(* delete old files and delete oldest files if number of files exceeds specified number *)
PROGRAM C09_MaintainFolders
VAR
	tArchiveCheck				: TIME := t#4s;
	fbMaintainArchive			: FB_PulseGenerator;
	tDeleteTimeCheck			: TIME := t#20m;
	fbMaintainDeleteTime		: FB_PulseGenerator;
	tClearProcessFolders		: TIME := T#500MS;
	tofClearProcessFolders		: TOF;
	
	nActivateBitWord			: DWORD; (* if index increase 32 bits it is necceasry to declar 64 bits var like LREAL;*)

	aMaintainFolders			: ARRAY[1..18] OF NT_StartProcess;
	aManualMaintain				: ARRAY[1..18] OF BOOL;

	fbMoveCHMToArchive			: FB_CHM_MoveToArchive;
	bZipCHMArchive				: BOOL;
	rtrigZipAfetrPassthrough	: R_TRIG;
	bManualZip					: BOOL;
	
(********************************************************************************
cMETS_CORE_FOLDERS					: ARRAY[1..cSYSTEM_FOLDER_LIMIT] OF T_FolderName :=[
			(*01*)'CHM\',		(*02*)'CHM\Archive\',		(*03*)'CHM\Error\',		(*04*)'CHM\OK\',		(*05*)'CHM\Commissioning_Mode\',	(*06*)'CHM\Restore\',
			(*07*)'PCM\',		(*08*)'PCM\Archive\',		(*09*)'PCM\Error\',		(*10*)'PCM\Incoming\',
			(*11*)'Settings\',	(*12*)'Settings\Backups\',	(*13*)'Settings\Recipe\',
			(*14*)'Cameras\',
			(*15*)'Printers\',	(*16*)'Printers\Templates'];
			
cMETS_AUX_FOLDERS					: ARRAY[1..cSYSTEM_FOLDER_LIMIT] OF T_FolderName :=[
			(*01*)'CAC\',		(*02*)'CAC\Archive\',		(*03*)'CAC\Error\',		(*04*)'CAC\Restored\',
			(*05*)'OAC\',		(*06*)'OAC\Error\',			(*07*)'OAC\Empty\',
			(*08*)'OCV\',		(*09*)'OCV\Error\',			(*10*)'OCV\Empty\',
			(*11*)'SystemLog\',
			(*12*)'ArchiveDB\',
			(*13*)'BridgeApp\Bridge_Core\',
			(*14*)'LoggerApp\Service\',
			(*15*)'WebHMI\',
			(*16*)'DeleteArchiveTool\'];

*************************************************************************************)
(********************************************************************************
Delete Items
	DeleteItem <path> <filesToKeep> [createLog] [deleteDirs] [dirsToKeep]
	path: Directory path
	filesToKeep: Number OF files TO RETAIN
	createLog: (Optional) Boolean to enable logging
	deleteDirs: (Optional) Boolean to include directories
	dirsToKeep: (Optional) Number of directories to retain

Delete by Time
	DeleteTime <path> <fileAge> [createLog] [deleteDirs] [ageUnit]
	path: Directory path
	fileAge: Maximum age of files to retain
	createLog: (Optional) Boolean to enable logging
	deleteDirs: (Optional) Boolean to include inside directories for file search
	ageUnit: (Optional) Time unit for age values (Day/Hour/Minute), defaults to Day

Archive
	Archive <chmArchiveFolder> <lastArchiveDateName> [createLog]
	chmArchiveFolder: Archive folder path
	lastArchiveDateName: Last archive date identifier
	createLog: (Optional) Boolean TO enable logging
*************************************************************************************)
END_VAR

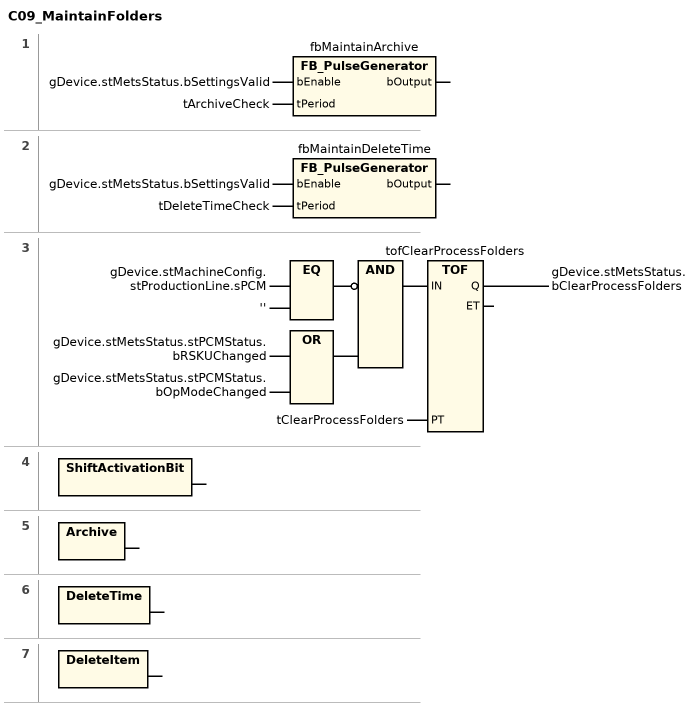
// NETWORK 1
fbMaintainArchive(bEnable := gDevice.stMetsStatus.bSettingsValid, tPeriod := tArchiveCheck); // FB_PulseGenerator

// NETWORK 2
fbMaintainDeleteTime(bEnable := gDevice.stMetsStatus.bSettingsValid, tPeriod := tDeleteTimeCheck); // FB_PulseGenerator

// NETWORK 3
tofClearProcessFolders(IN := NOT (gDevice.stMachineConfig.stProductionLine.sPCM = '') AND (gDevice.stMetsStatus.stPCMStatus.bRSKUChanged OR gDevice.stMetsStatus.stPCMStatus.bOpModeChanged), PT := tClearProcessFolders); // TOF
gDevice.stMetsStatus.bClearProcessFolders := tofClearProcessFolders.Q;

// NETWORK 4
ShiftActivationBit();

// NETWORK 5
Archive();

// NETWORK 6
DeleteTime();

// NETWORK 7
DeleteItem();

ACTION Archive:
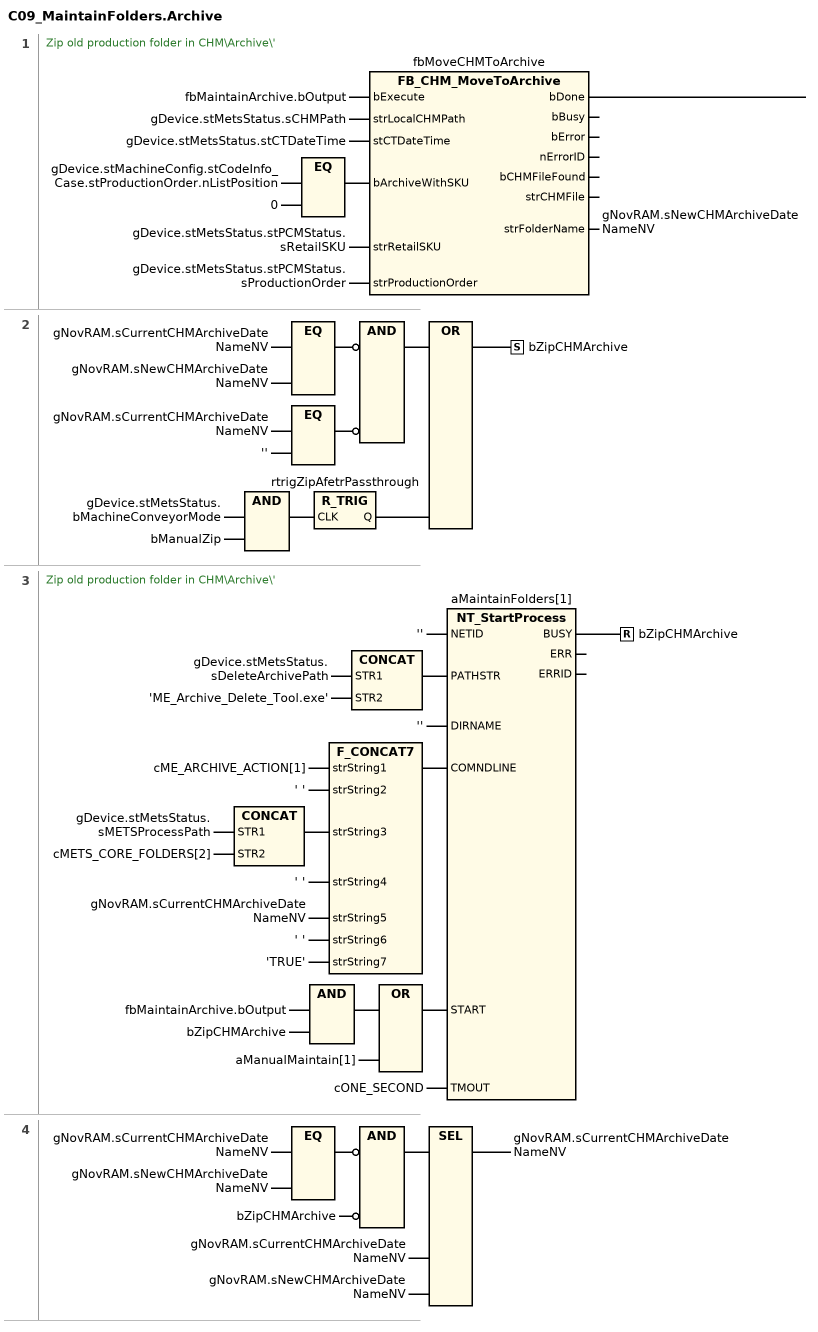
// NETWORK 1
// 					Zip old production folder in CHM\Archive\'
//
//
fbMoveCHMToArchive(
    bExecute := fbMaintainArchive.bOutput,
    strLocalCHMPath := gDevice.stMetsStatus.sCHMPath,
    stCTDateTime := gDevice.stMetsStatus.stCTDateTime,
    bArchiveWithSKU := gDevice.stMachineConfig.stCodeInfo_Case.stProductionOrder.nListPosition = 0,
    strRetailSKU := gDevice.stMetsStatus.stPCMStatus.sRetailSKU,
    strProductionOrder := gDevice.stMetsStatus.stPCMStatus.sProductionOrder,
    strFolderName => gNovRAM.sNewCHMArchiveDateNameNV); // FB_CHM_MoveToArchive

// NETWORK 2
rtrigZipAfetrPassthrough(CLK := gDevice.stMetsStatus.bMachineConveyorMode AND bManualZip); // R_TRIG
bZipCHMArchive S= NOT (gNovRAM.sCurrentCHMArchiveDateNameNV = gNovRAM.sNewCHMArchiveDateNameNV) AND NOT (gNovRAM.sCurrentCHMArchiveDateNameNV = '') OR rtrigZipAfetrPassthrough.Q;

// NETWORK 3
// Zip old production folder in CHM\Archive\'
aMaintainFolders[1](
    NETID := '',
    PATHSTR := CONCAT(STR1 := gDevice.stMetsStatus.sDeleteArchivePath, STR2 := 'ME_Archive_Delete_Tool.exe'),
    DIRNAME := '',
    COMNDLINE := F_CONCAT7(strString1 := cME_ARCHIVE_ACTION[1], strString2 := ' ', strString3 := CONCAT(STR1 := gDevice.stMetsStatus.sMETSProcessPath, STR2 := cMETS_CORE_FOLDERS[2]), strString4 := ' ', strString5 := gNovRAM.sCurrentCHMArchiveDateNameNV, strString6 := ' ', strString7 := 'TRUE'),
    START := fbMaintainArchive.bOutput AND bZipCHMArchive OR aManualMaintain[1],
    TMOUT := cONE_SECOND); // NT_StartProcess
bZipCHMArchive R= aMaintainFolders[1].BUSY;

// NETWORK 4
gNovRAM.sCurrentCHMArchiveDateNameNV := SEL(NOT (gNovRAM.sCurrentCHMArchiveDateNameNV = gNovRAM.sNewCHMArchiveDateNameNV) AND NOT bZipCHMArchive, gNovRAM.sCurrentCHMArchiveDateNameNV, gNovRAM.sNewCHMArchiveDateNameNV);
END_ACTION

ACTION DeleteItem:
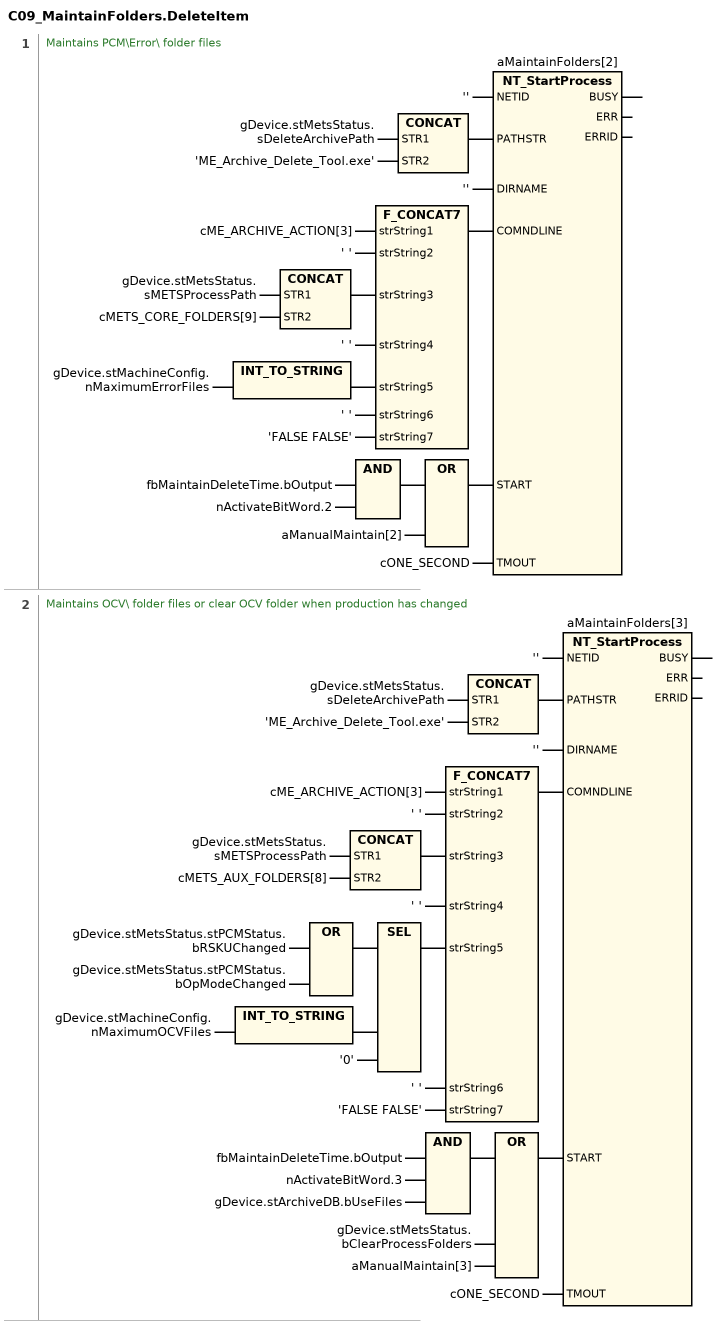
// NETWORK 1
// Maintains PCM\Error\ folder files
aMaintainFolders[2](
    NETID := '',
    PATHSTR := CONCAT(STR1 := gDevice.stMetsStatus.sDeleteArchivePath, STR2 := 'ME_Archive_Delete_Tool.exe'),
    DIRNAME := '',
    COMNDLINE := F_CONCAT7(strString1 := cME_ARCHIVE_ACTION[3], strString2 := ' ', strString3 := CONCAT(STR1 := gDevice.stMetsStatus.sMETSProcessPath, STR2 := cMETS_CORE_FOLDERS[9]), strString4 := ' ', strString5 := INT_TO_STRING(gDevice.stMachineConfig.nMaximumErrorFiles), strString6 := ' ', strString7 := 'FALSE FALSE'),
    START := fbMaintainDeleteTime.bOutput AND nActivateBitWord.2 OR aManualMaintain[2],
    TMOUT := cONE_SECOND); // NT_StartProcess

// NETWORK 2
// Maintains OCV\ folder files or clear OCV folder when production has changed
aMaintainFolders[3](
    NETID := '',
    PATHSTR := CONCAT(STR1 := gDevice.stMetsStatus.sDeleteArchivePath, STR2 := 'ME_Archive_Delete_Tool.exe'),
    DIRNAME := '',
    COMNDLINE := F_CONCAT7(strString1 := cME_ARCHIVE_ACTION[3], strString2 := ' ', strString3 := CONCAT(STR1 := gDevice.stMetsStatus.sMETSProcessPath, STR2 := cMETS_AUX_FOLDERS[8]), strString4 := ' ', strString5 := SEL(gDevice.stMetsStatus.stPCMStatus.bRSKUChanged OR gDevice.stMetsStatus.stPCMStatus.bOpModeChanged, INT_TO_STRING(gDevice.stMachineConfig.nMaximumOCVFiles), '0'), strString6 := ' ', strString7 := 'FALSE FALSE'),
    START := fbMaintainDeleteTime.bOutput AND nActivateBitWord.3 AND gDevice.stArchiveDB.bUseFiles OR gDevice.stMetsStatus.bClearProcessFolders OR aManualMaintain[3],
    TMOUT := cONE_SECOND); // NT_StartProcess

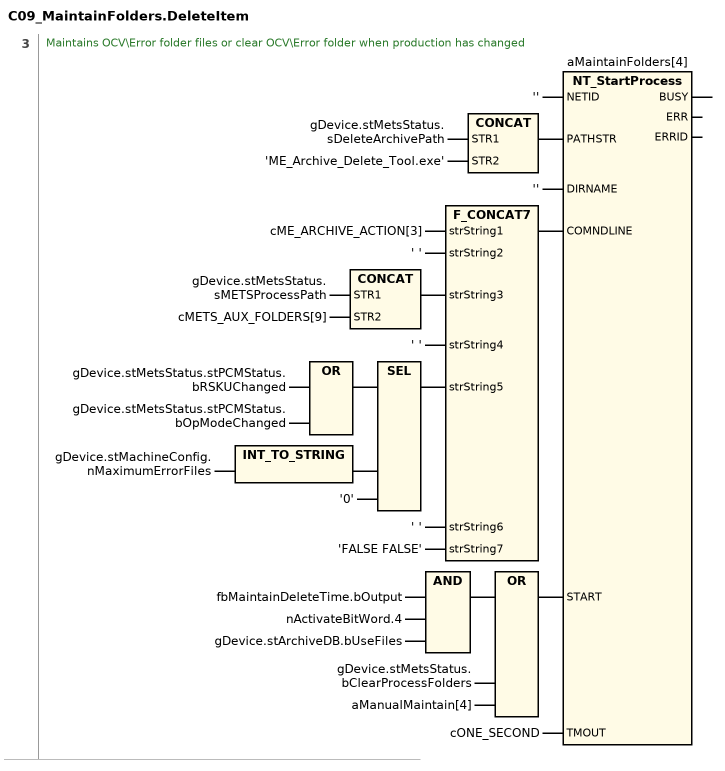
// NETWORK 3
// Maintains OCV\Error folder files or clear OCV\Error folder when production has changed
aMaintainFolders[4](
    NETID := '',
    PATHSTR := CONCAT(STR1 := gDevice.stMetsStatus.sDeleteArchivePath, STR2 := 'ME_Archive_Delete_Tool.exe'),
    DIRNAME := '',
    COMNDLINE := F_CONCAT7(strString1 := cME_ARCHIVE_ACTION[3], strString2 := ' ', strString3 := CONCAT(STR1 := gDevice.stMetsStatus.sMETSProcessPath, STR2 := cMETS_AUX_FOLDERS[9]), strString4 := ' ', strString5 := SEL(gDevice.stMetsStatus.stPCMStatus.bRSKUChanged OR gDevice.stMetsStatus.stPCMStatus.bOpModeChanged, INT_TO_STRING(gDevice.stMachineConfig.nMaximumErrorFiles), '0'), strString6 := ' ', strString7 := 'FALSE FALSE'),
    START := fbMaintainDeleteTime.bOutput AND nActivateBitWord.4 AND gDevice.stArchiveDB.bUseFiles OR gDevice.stMetsStatus.bClearProcessFolders OR aManualMaintain[4],
    TMOUT := cONE_SECOND); // NT_StartProcess

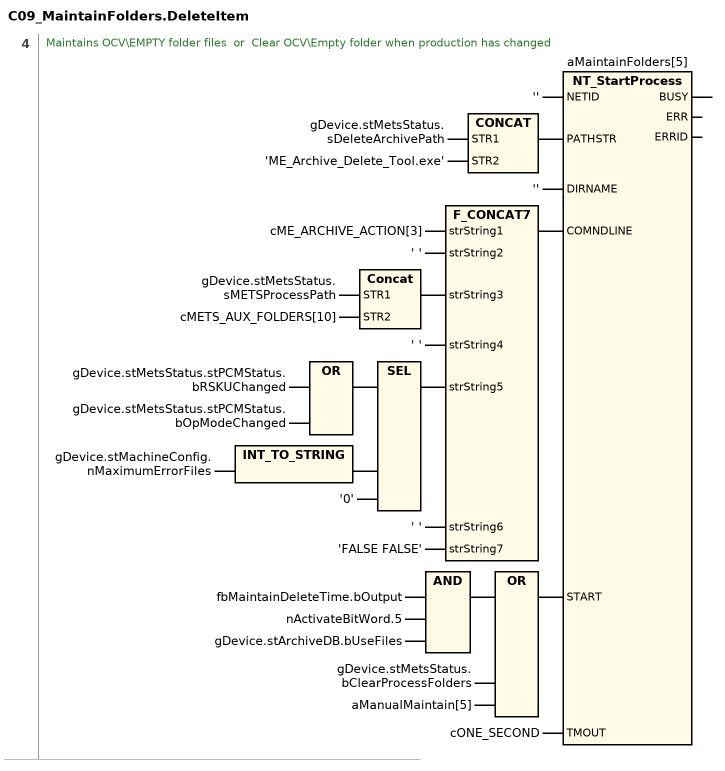
// NETWORK 4
// Maintains OCV\EMPTY folder files  or  Clear OCV\Empty folder when production has changed
aMaintainFolders[5](
    NETID := '',
    PATHSTR := CONCAT(STR1 := gDevice.stMetsStatus.sDeleteArchivePath, STR2 := 'ME_Archive_Delete_Tool.exe'),
    DIRNAME := '',
    COMNDLINE := F_CONCAT7(strString1 := cME_ARCHIVE_ACTION[3], strString2 := ' ', strString3 := Concat(STR1 := gDevice.stMetsStatus.sMETSProcessPath, STR2 := cMETS_AUX_FOLDERS[10]), strString4 := ' ', strString5 := SEL(gDevice.stMetsStatus.stPCMStatus.bRSKUChanged OR gDevice.stMetsStatus.stPCMStatus.bOpModeChanged, INT_TO_STRING(gDevice.stMachineConfig.nMaximumErrorFiles), '0'), strString6 := ' ', strString7 := 'FALSE FALSE'),
    START := fbMaintainDeleteTime.bOutput AND nActivateBitWord.5 AND gDevice.stArchiveDB.bUseFiles OR gDevice.stMetsStatus.bClearProcessFolders OR aManualMaintain[5],
    TMOUT := cONE_SECOND); // NT_StartProcess

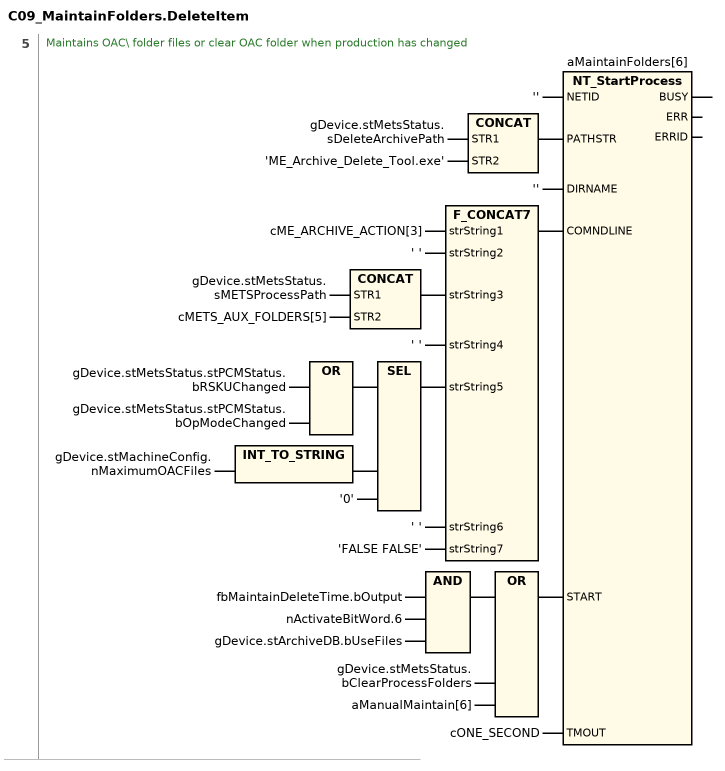
// NETWORK 5
// Maintains OAC\ folder files or clear OAC folder when production has changed
aMaintainFolders[6](
    NETID := '',
    PATHSTR := CONCAT(STR1 := gDevice.stMetsStatus.sDeleteArchivePath, STR2 := 'ME_Archive_Delete_Tool.exe'),
    DIRNAME := '',
    COMNDLINE := F_CONCAT7(strString1 := cME_ARCHIVE_ACTION[3], strString2 := ' ', strString3 := CONCAT(STR1 := gDevice.stMetsStatus.sMETSProcessPath, STR2 := cMETS_AUX_FOLDERS[5]), strString4 := ' ', strString5 := SEL(gDevice.stMetsStatus.stPCMStatus.bRSKUChanged OR gDevice.stMetsStatus.stPCMStatus.bOpModeChanged, INT_TO_STRING(gDevice.stMachineConfig.nMaximumOACFiles), '0'), strString6 := ' ', strString7 := 'FALSE FALSE'),
    START := fbMaintainDeleteTime.bOutput AND nActivateBitWord.6 AND gDevice.stArchiveDB.bUseFiles OR gDevice.stMetsStatus.bClearProcessFolders OR aManualMaintain[6],
    TMOUT := cONE_SECOND); // NT_StartProcess

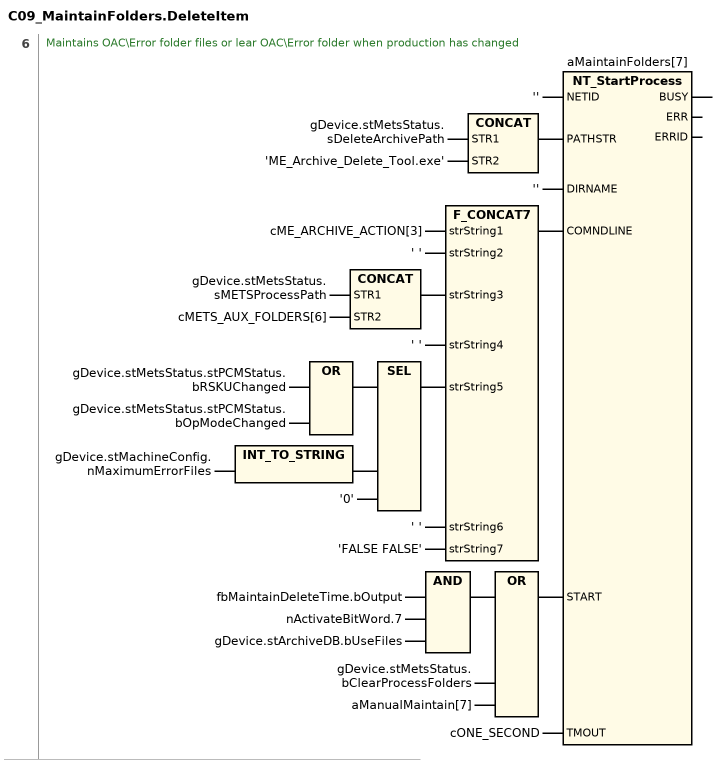
// NETWORK 6
// Maintains OAC\Error folder files or lear OAC\Error folder when production has changed
aMaintainFolders[7](
    NETID := '',
    PATHSTR := CONCAT(STR1 := gDevice.stMetsStatus.sDeleteArchivePath, STR2 := 'ME_Archive_Delete_Tool.exe'),
    DIRNAME := '',
    COMNDLINE := F_CONCAT7(strString1 := cME_ARCHIVE_ACTION[3], strString2 := ' ', strString3 := CONCAT(STR1 := gDevice.stMetsStatus.sMETSProcessPath, STR2 := cMETS_AUX_FOLDERS[6]), strString4 := ' ', strString5 := SEL(gDevice.stMetsStatus.stPCMStatus.bRSKUChanged OR gDevice.stMetsStatus.stPCMStatus.bOpModeChanged, INT_TO_STRING(gDevice.stMachineConfig.nMaximumErrorFiles), '0'), strString6 := ' ', strString7 := 'FALSE FALSE'),
    START := fbMaintainDeleteTime.bOutput AND nActivateBitWord.7 AND gDevice.stArchiveDB.bUseFiles OR gDevice.stMetsStatus.bClearProcessFolders OR aManualMaintain[7],
    TMOUT := cONE_SECOND); // NT_StartProcess

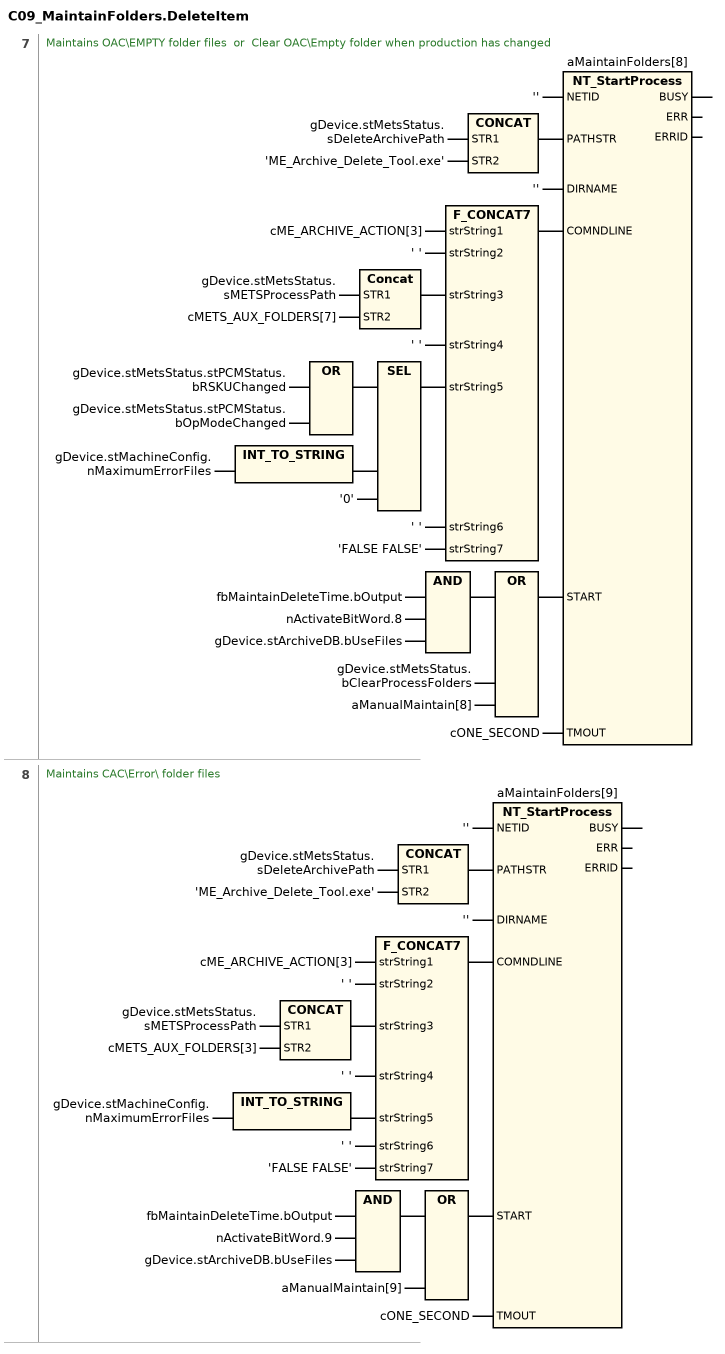
// NETWORK 7
// Maintains OAC\EMPTY folder files  or  Clear OAC\Empty folder when production has changed
aMaintainFolders[8](
    NETID := '',
    PATHSTR := CONCAT(STR1 := gDevice.stMetsStatus.sDeleteArchivePath, STR2 := 'ME_Archive_Delete_Tool.exe'),
    DIRNAME := '',
    COMNDLINE := F_CONCAT7(strString1 := cME_ARCHIVE_ACTION[3], strString2 := ' ', strString3 := Concat(STR1 := gDevice.stMetsStatus.sMETSProcessPath, STR2 := cMETS_AUX_FOLDERS[7]), strString4 := ' ', strString5 := SEL(gDevice.stMetsStatus.stPCMStatus.bRSKUChanged OR gDevice.stMetsStatus.stPCMStatus.bOpModeChanged, INT_TO_STRING(gDevice.stMachineConfig.nMaximumErrorFiles), '0'), strString6 := ' ', strString7 := 'FALSE FALSE'),
    START := fbMaintainDeleteTime.bOutput AND nActivateBitWord.8 AND gDevice.stArchiveDB.bUseFiles OR gDevice.stMetsStatus.bClearProcessFolders OR aManualMaintain[8],
    TMOUT := cONE_SECOND); // NT_StartProcess

// NETWORK 8
// Maintains CAC\Error\ folder files
aMaintainFolders[9](
    NETID := '',
    PATHSTR := CONCAT(STR1 := gDevice.stMetsStatus.sDeleteArchivePath, STR2 := 'ME_Archive_Delete_Tool.exe'),
    DIRNAME := '',
    COMNDLINE := F_CONCAT7(strString1 := cME_ARCHIVE_ACTION[3], strString2 := ' ', strString3 := CONCAT(STR1 := gDevice.stMetsStatus.sMETSProcessPath, STR2 := cMETS_AUX_FOLDERS[3]), strString4 := ' ', strString5 := INT_TO_STRING(gDevice.stMachineConfig.nMaximumErrorFiles), strString6 := ' ', strString7 := 'FALSE FALSE'),
    START := fbMaintainDeleteTime.bOutput AND nActivateBitWord.9 AND gDevice.stArchiveDB.bUseFiles OR aManualMaintain[9],
    TMOUT := cONE_SECOND); // NT_StartProcess

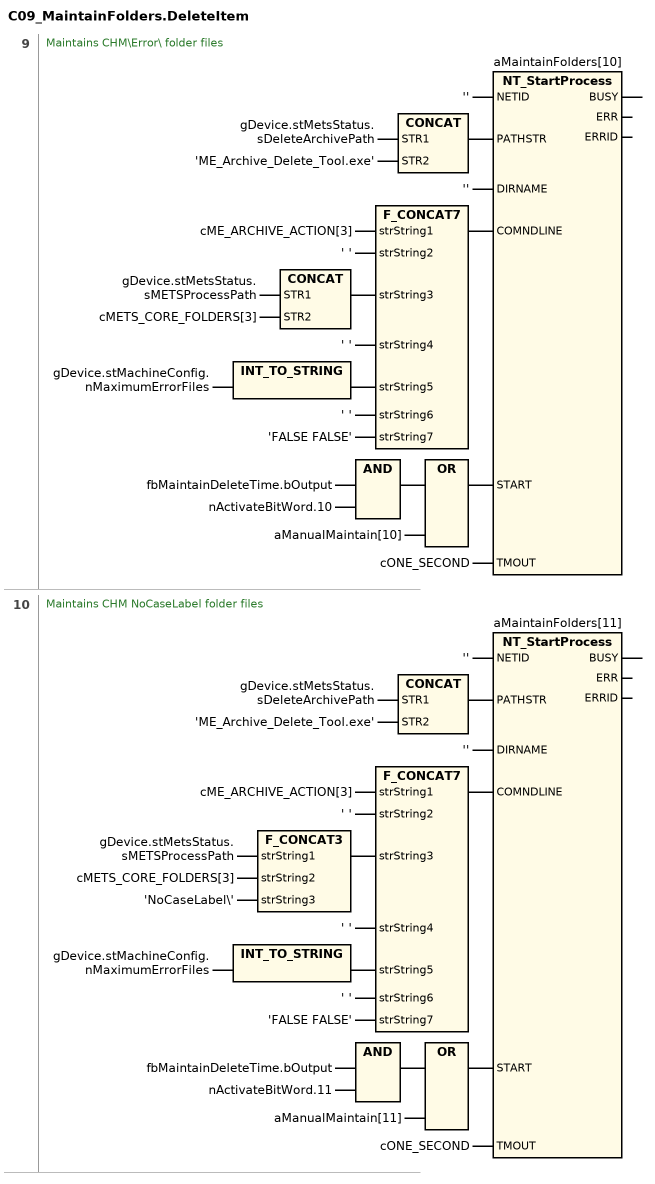
// NETWORK 9
// Maintains CHM\Error\ folder files
aMaintainFolders[10](
    NETID := '',
    PATHSTR := CONCAT(STR1 := gDevice.stMetsStatus.sDeleteArchivePath, STR2 := 'ME_Archive_Delete_Tool.exe'),
    DIRNAME := '',
    COMNDLINE := F_CONCAT7(strString1 := cME_ARCHIVE_ACTION[3], strString2 := ' ', strString3 := CONCAT(STR1 := gDevice.stMetsStatus.sMETSProcessPath, STR2 := cMETS_CORE_FOLDERS[3]), strString4 := ' ', strString5 := INT_TO_STRING(gDevice.stMachineConfig.nMaximumErrorFiles), strString6 := ' ', strString7 := 'FALSE FALSE'),
    START := fbMaintainDeleteTime.bOutput AND nActivateBitWord.10 OR aManualMaintain[10],
    TMOUT := cONE_SECOND); // NT_StartProcess

// NETWORK 10
// Maintains CHM NoCaseLabel folder files
aMaintainFolders[11](
    NETID := '',
    PATHSTR := CONCAT(STR1 := gDevice.stMetsStatus.sDeleteArchivePath, STR2 := 'ME_Archive_Delete_Tool.exe'),
    DIRNAME := '',
    COMNDLINE := F_CONCAT7(strString1 := cME_ARCHIVE_ACTION[3], strString2 := ' ', strString3 := F_CONCAT3(strString1 := gDevice.stMetsStatus.sMETSProcessPath, strString2 := cMETS_CORE_FOLDERS[3], strString3 := 'NoCaseLabel\'), strString4 := ' ', strString5 := INT_TO_STRING(gDevice.stMachineConfig.nMaximumErrorFiles), strString6 := ' ', strString7 := 'FALSE FALSE'),
    START := fbMaintainDeleteTime.bOutput AND nActivateBitWord.11 OR aManualMaintain[11],
    TMOUT := cONE_SECOND); // NT_StartProcess
END_ACTION

ACTION DeleteTime:
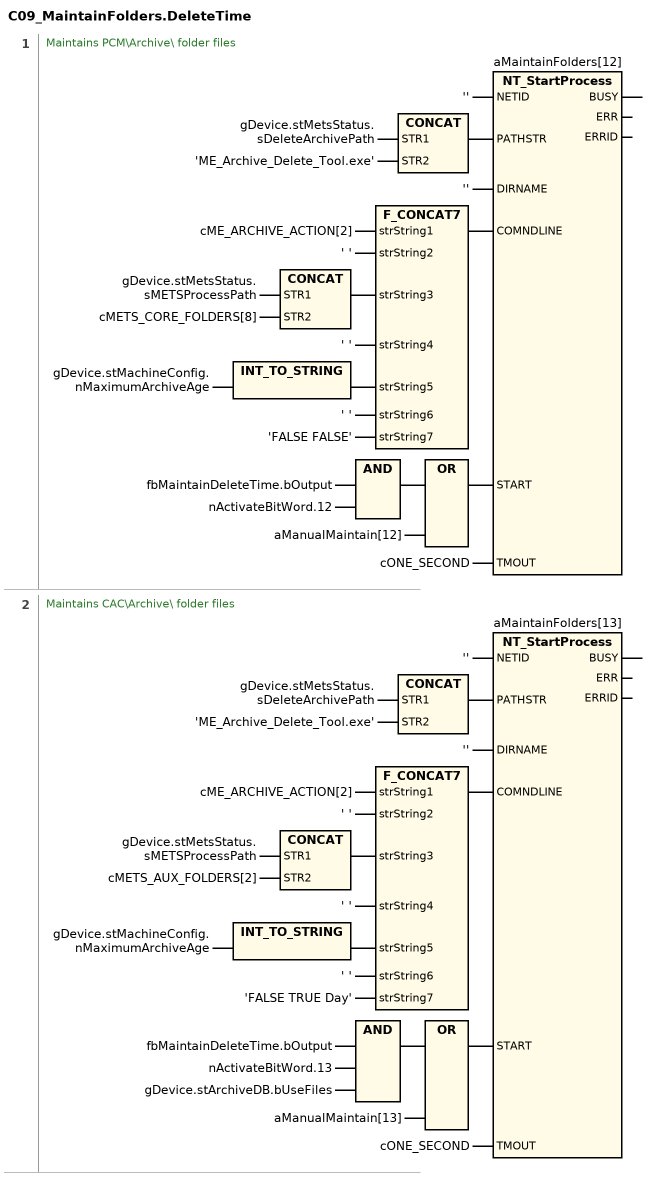
// NETWORK 1
// Maintains PCM\Archive\ folder files
aMaintainFolders[12](
    NETID := '',
    PATHSTR := CONCAT(STR1 := gDevice.stMetsStatus.sDeleteArchivePath, STR2 := 'ME_Archive_Delete_Tool.exe'),
    DIRNAME := '',
    COMNDLINE := F_CONCAT7(strString1 := cME_ARCHIVE_ACTION[2], strString2 := ' ', strString3 := CONCAT(STR1 := gDevice.stMetsStatus.sMETSProcessPath, STR2 := cMETS_CORE_FOLDERS[8]), strString4 := ' ', strString5 := INT_TO_STRING(gDevice.stMachineConfig.nMaximumArchiveAge), strString6 := ' ', strString7 := 'FALSE FALSE'),
    START := fbMaintainDeleteTime.bOutput AND nActivateBitWord.12 OR aManualMaintain[12],
    TMOUT := cONE_SECOND); // NT_StartProcess

// NETWORK 2
// Maintains CAC\Archive\ folder files
aMaintainFolders[13](
    NETID := '',
    PATHSTR := CONCAT(STR1 := gDevice.stMetsStatus.sDeleteArchivePath, STR2 := 'ME_Archive_Delete_Tool.exe'),
    DIRNAME := '',
    COMNDLINE := F_CONCAT7(strString1 := cME_ARCHIVE_ACTION[2], strString2 := ' ', strString3 := CONCAT(STR1 := gDevice.stMetsStatus.sMETSProcessPath, STR2 := cMETS_AUX_FOLDERS[2]), strString4 := ' ', strString5 := INT_TO_STRING(gDevice.stMachineConfig.nMaximumArchiveAge), strString6 := ' ', strString7 := 'FALSE TRUE Day'),
    START := fbMaintainDeleteTime.bOutput AND nActivateBitWord.13 AND gDevice.stArchiveDB.bUseFiles OR aManualMaintain[13],
    TMOUT := cONE_SECOND); // NT_StartProcess

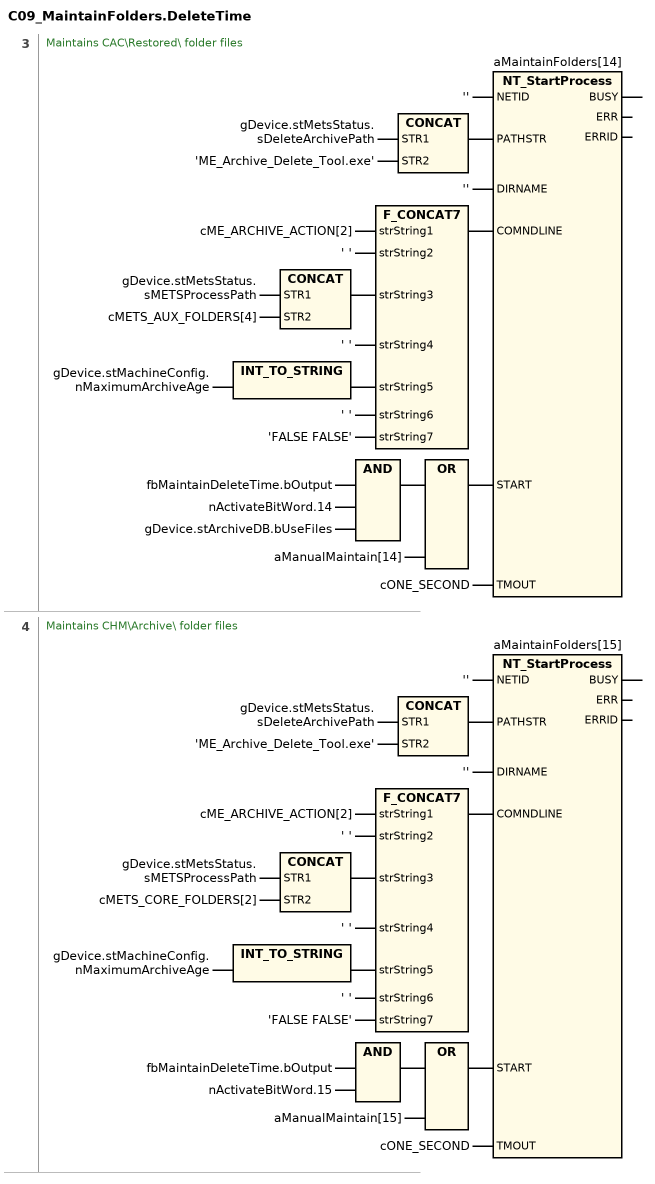
// NETWORK 3
// Maintains CAC\Restored\ folder files
aMaintainFolders[14](
    NETID := '',
    PATHSTR := CONCAT(STR1 := gDevice.stMetsStatus.sDeleteArchivePath, STR2 := 'ME_Archive_Delete_Tool.exe'),
    DIRNAME := '',
    COMNDLINE := F_CONCAT7(strString1 := cME_ARCHIVE_ACTION[2], strString2 := ' ', strString3 := CONCAT(STR1 := gDevice.stMetsStatus.sMETSProcessPath, STR2 := cMETS_AUX_FOLDERS[4]), strString4 := ' ', strString5 := INT_TO_STRING(gDevice.stMachineConfig.nMaximumArchiveAge), strString6 := ' ', strString7 := 'FALSE FALSE'),
    START := fbMaintainDeleteTime.bOutput AND nActivateBitWord.14 AND gDevice.stArchiveDB.bUseFiles OR aManualMaintain[14],
    TMOUT := cONE_SECOND); // NT_StartProcess

// NETWORK 4
// Maintains CHM\Archive\ folder files
aMaintainFolders[15](
    NETID := '',
    PATHSTR := CONCAT(STR1 := gDevice.stMetsStatus.sDeleteArchivePath, STR2 := 'ME_Archive_Delete_Tool.exe'),
    DIRNAME := '',
    COMNDLINE := F_CONCAT7(strString1 := cME_ARCHIVE_ACTION[2], strString2 := ' ', strString3 := CONCAT(STR1 := gDevice.stMetsStatus.sMETSProcessPath, STR2 := cMETS_CORE_FOLDERS[2]), strString4 := ' ', strString5 := INT_TO_STRING(gDevice.stMachineConfig.nMaximumArchiveAge), strString6 := ' ', strString7 := 'FALSE FALSE'),
    START := fbMaintainDeleteTime.bOutput AND nActivateBitWord.15 OR aManualMaintain[15],
    TMOUT := cONE_SECOND); // NT_StartProcess

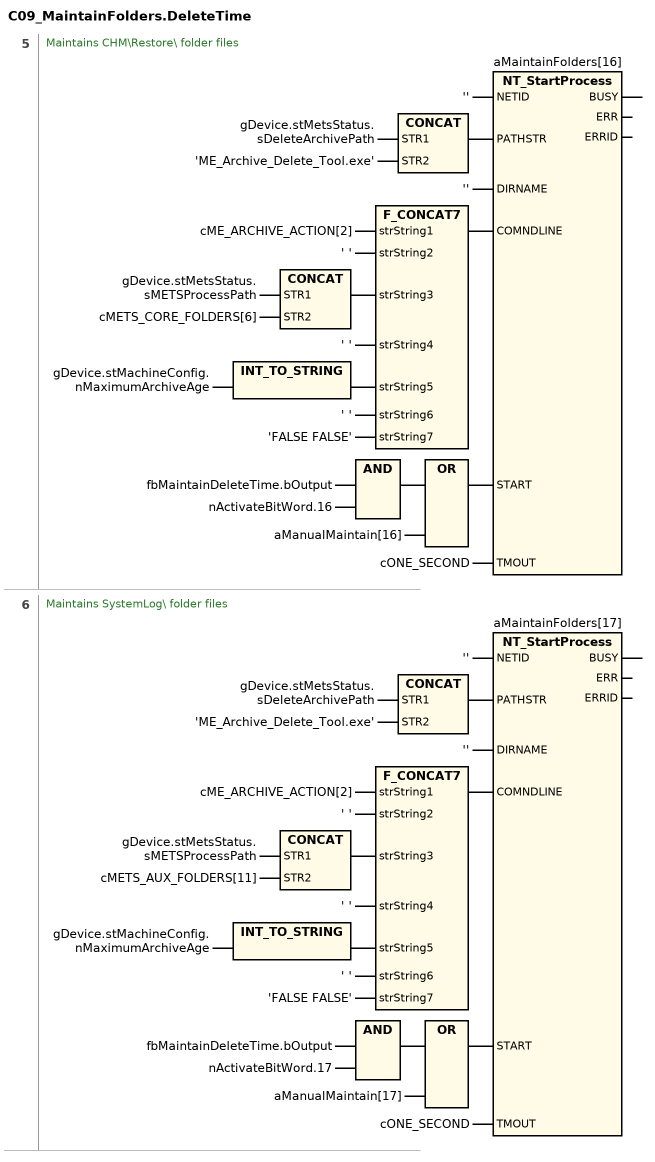
// NETWORK 5
// Maintains CHM\Restore\ folder files
aMaintainFolders[16](
    NETID := '',
    PATHSTR := CONCAT(STR1 := gDevice.stMetsStatus.sDeleteArchivePath, STR2 := 'ME_Archive_Delete_Tool.exe'),
    DIRNAME := '',
    COMNDLINE := F_CONCAT7(strString1 := cME_ARCHIVE_ACTION[2], strString2 := ' ', strString3 := CONCAT(STR1 := gDevice.stMetsStatus.sMETSProcessPath, STR2 := cMETS_CORE_FOLDERS[6]), strString4 := ' ', strString5 := INT_TO_STRING(gDevice.stMachineConfig.nMaximumArchiveAge), strString6 := ' ', strString7 := 'FALSE FALSE'),
    START := fbMaintainDeleteTime.bOutput AND nActivateBitWord.16 OR aManualMaintain[16],
    TMOUT := cONE_SECOND); // NT_StartProcess

// NETWORK 6
// Maintains SystemLog\ folder files
aMaintainFolders[17](
    NETID := '',
    PATHSTR := CONCAT(STR1 := gDevice.stMetsStatus.sDeleteArchivePath, STR2 := 'ME_Archive_Delete_Tool.exe'),
    DIRNAME := '',
    COMNDLINE := F_CONCAT7(strString1 := cME_ARCHIVE_ACTION[2], strString2 := ' ', strString3 := CONCAT(STR1 := gDevice.stMetsStatus.sMETSProcessPath, STR2 := cMETS_AUX_FOLDERS[11]), strString4 := ' ', strString5 := INT_TO_STRING(gDevice.stMachineConfig.nMaximumArchiveAge), strString6 := ' ', strString7 := 'FALSE FALSE'),
    START := fbMaintainDeleteTime.bOutput AND nActivateBitWord.17 OR aManualMaintain[17],
    TMOUT := cONE_SECOND); // NT_StartProcess

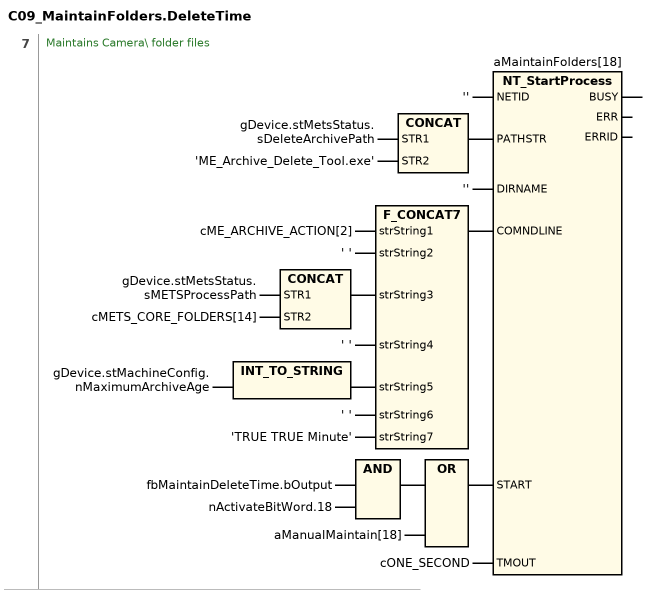
// NETWORK 7
// Maintains Camera\ folder files
aMaintainFolders[18](
    NETID := '',
    PATHSTR := CONCAT(STR1 := gDevice.stMetsStatus.sDeleteArchivePath, STR2 := 'ME_Archive_Delete_Tool.exe'),
    DIRNAME := '',
    COMNDLINE := F_CONCAT7(strString1 := cME_ARCHIVE_ACTION[2], strString2 := ' ', strString3 := CONCAT(STR1 := gDevice.stMetsStatus.sMETSProcessPath, STR2 := cMETS_CORE_FOLDERS[14]), strString4 := ' ', strString5 := INT_TO_STRING(gDevice.stMachineConfig.nMaximumArchiveAge), strString6 := ' ', strString7 := 'TRUE TRUE Minute'),
    START := fbMaintainDeleteTime.bOutput AND nActivateBitWord.18 OR aManualMaintain[18],
    TMOUT := cONE_SECOND); // NT_StartProcess
END_ACTION

ACTION ShiftActivationBit:
IF fbMaintainDeleteTime.bOutput	THEN
	IF nActivateBitWord = 0 THEN
		nActivateBitWord := 1;
	ELSE
		nActivateBitWord :=SHL(nActivateBitWord,1);
	END_IF
END_IF
END_ACTION

END_PROGRAM

(* stored: Version 1.1.0.1
   POU C09_MaintainFolders: Id {b89b74f7-3658-4720-addf-2afb9a9065cd}, SpecialFunc None
   Action Archive: Id {b51be478-c4ea-481c-ad6e-ebbe95254e6a}
   Action DeleteItem: Id {f8ec7b99-6612-4740-9c03-3e45dca7fc99}
   Action DeleteTime: Id {960aca6a-468c-4531-b56a-c74dc626c107}
   Action ShiftActivationBit: Id {a10af811-c787-4570-8da7-7a0544dfed28} *)
